{attribute 'qualified_only'}
{attribute 'strict'}
TYPE E_Mode :
(
	enum_member := 0
);
END_TYPE

(* stored: Version 1.1.0.1, ProductVersion 3.1.4024.10
   DUT E_Mode: Id {f8d1d1e2-5a74-4efa-a324-8b73d4f6144f} *)
